VAR_GLOBAL 
	stToRobot1	: DUT_SysToRobot1; //
	stFromRobot1  : DUT_SysFromRobot1; //
END_VAR

(* stored: Version 1.1.0.1, ProductVersion 3.1.4024.9
   GVL GVL_Robot: Id {567953b5-67db-4a2c-bd18-7d05a2720581} *)
